(* IEC 61131-3 sources: stc/tests/conveyor, 2 files *)

(* ---- conveyor.st ---- *)
(* Conveyor Belt Control Function Block
   Models a 3-zone conveyor with photoeye sensors, jam detection,
   and state-machine sequencing.

   States:
     0 = IDLE      - Waiting for product
     1 = RUNNING   - Conveyor moving, product in transit
     2 = JAM       - Sensor blocked too long, fault
     3 = STOPPED   - Operator stop requested
*)

FUNCTION_BLOCK ConveyorZone
VAR_INPUT
    Enable      : BOOL;      (* Master enable *)
    SensorEntry : BOOL;      (* Photoeye at zone entry *)
    SensorExit  : BOOL;      (* Photoeye at zone exit *)
    Reset       : BOOL;      (* Reset from jam fault *)
    JamTimeLimit : TIME := T#10s;  (* Max time sensor can be blocked *)
END_VAR

VAR_OUTPUT
    MotorFwd    : BOOL;      (* Drive motor forward *)
    ZoneOccupied : BOOL;     (* Product present in zone *)
    JamFault    : BOOL;      (* Jam detected *)
    State       : INT;       (* Current state *)
    ProductCount : DINT;     (* Products that have exited *)
END_VAR

VAR
    JamTimer    : TON;       (* Jam detection timer *)
    ExitEdge    : R_TRIG;    (* Detects product leaving zone *)
    EntryEdge   : R_TRIG;    (* Detects product entering zone *)
    Counter     : CTU;       (* Product counter *)
END_VAR

    (* Detect product entry and exit edges *)
    EntryEdge(CLK := SensorEntry);
    ExitEdge(CLK := NOT SensorExit);  (* Photoeye: TRUE = blocked *)

    (* State machine *)
    CASE State OF
        0: (* IDLE *)
            MotorFwd := FALSE;
            IF Enable AND SensorEntry THEN
                State := 1;
                ZoneOccupied := TRUE;
            END_IF;

        1: (* RUNNING *)
            MotorFwd := TRUE;
            (* Check for product exit *)
            IF NOT SensorEntry AND NOT SensorExit THEN
                ZoneOccupied := FALSE;
                Counter(CU := TRUE, R := FALSE, PV := 9999);
                State := 0;
            END_IF;
            (* Check for jam *)
            JamTimer(IN := SensorEntry, PT := JamTimeLimit);
            IF JamTimer.Q THEN
                State := 2;
            END_IF;
            IF NOT Enable THEN
                State := 3;
            END_IF;

        2: (* JAM *)
            MotorFwd := FALSE;
            JamFault := TRUE;
            IF Reset THEN
                JamFault := FALSE;
                JamTimer(IN := FALSE, PT := JamTimeLimit);
                State := 0;
            END_IF;

        3: (* STOPPED *)
            MotorFwd := FALSE;
            IF Enable THEN
                State := 1;
            END_IF;
    END_CASE;

    ProductCount := Counter.CV;

    (* Reset counter edge *)
    Counter(CU := FALSE, R := FALSE, PV := 9999);
END_FUNCTION_BLOCK

(* ---- conveyor_test.st ---- *)
(* Conveyor Belt Test Suite
   Tests state machine transitions, jam detection, product counting,
   and enable/disable behavior for a 3-zone conveyor system.
*)

TEST_CASE 'Conveyor starts in IDLE state'
VAR
    State : INT := 0;
    MotorFwd : BOOL := FALSE;
END_VAR
    ASSERT_EQ(State, 0);
    ASSERT_FALSE(MotorFwd);
END_TEST_CASE

TEST_CASE 'Product entry transitions IDLE to RUNNING'
VAR
    State : INT := 0;
    Enable : BOOL := TRUE;
    SensorEntry : BOOL;
    MotorFwd : BOOL;
END_VAR
    (* No product yet *)
    SensorEntry := FALSE;
    CASE State OF
        0:
            MotorFwd := FALSE;
            IF Enable AND SensorEntry THEN
                State := 1;
            END_IF;
    END_CASE;
    ASSERT_EQ(State, 0);
    ASSERT_FALSE(MotorFwd);

    (* Product arrives *)
    SensorEntry := TRUE;
    CASE State OF
        0:
            MotorFwd := FALSE;
            IF Enable AND SensorEntry THEN
                State := 1;
            END_IF;
    END_CASE;
    ASSERT_EQ(State, 1);
END_TEST_CASE

TEST_CASE 'Jam timer triggers fault after timeout'
VAR
    JamTimer : TON;
    SensorEntry : BOOL := TRUE;
    JamFault : BOOL;
END_VAR
    (* Sensor blocked, start timing *)
    JamTimer(IN := SensorEntry, PT := T#10s);
    ASSERT_FALSE(JamTimer.Q);

    (* 8 seconds pass, still no jam *)
    ADVANCE_TIME(T#8s);
    JamTimer(IN := SensorEntry, PT := T#10s);
    ASSERT_FALSE(JamTimer.Q);

    (* 3 more seconds, total 11s > 10s preset *)
    ADVANCE_TIME(T#3s);
    JamTimer(IN := SensorEntry, PT := T#10s);
    ASSERT_TRUE(JamTimer.Q);
    JamFault := JamTimer.Q;
    ASSERT_TRUE(JamFault);
END_TEST_CASE

TEST_CASE 'Jam resets on operator Reset signal'
VAR
    JamTimer : TON;
    JamFault : BOOL := TRUE;
    Reset : BOOL;
    State : INT := 2;
END_VAR
    (* In JAM state, operator presses reset *)
    Reset := TRUE;
    IF Reset THEN
        JamFault := FALSE;
        JamTimer(IN := FALSE, PT := T#10s);
        State := 0;
    END_IF;

    ASSERT_FALSE(JamFault);
    ASSERT_EQ(State, 0);
    ASSERT_FALSE(JamTimer.Q);
END_TEST_CASE

TEST_CASE 'Product counter increments on product exit'
VAR
    Counter : CTU;
END_VAR
    (* Simulate 3 products passing through *)
    Counter(CU := FALSE, R := FALSE, PV := 9999);

    (* Product 1 exits *)
    Counter(CU := TRUE, R := FALSE, PV := 9999);
    ASSERT_EQ(Counter.CV, 1);
    Counter(CU := FALSE, R := FALSE, PV := 9999);

    (* Product 2 exits *)
    Counter(CU := TRUE, R := FALSE, PV := 9999);
    ASSERT_EQ(Counter.CV, 2);
    Counter(CU := FALSE, R := FALSE, PV := 9999);

    (* Product 3 exits *)
    Counter(CU := TRUE, R := FALSE, PV := 9999);
    ASSERT_EQ(Counter.CV, 3);
    ASSERT_FALSE(Counter.Q);  (* PV=9999, far from reached *)
END_TEST_CASE

TEST_CASE 'Disable stops conveyor motor'
VAR
    State : INT := 1;  (* RUNNING *)
    Enable : BOOL;
    MotorFwd : BOOL := TRUE;
END_VAR
    (* Operator disables *)
    Enable := FALSE;

    CASE State OF
        1:
            IF NOT Enable THEN
                State := 3;
                MotorFwd := FALSE;
            END_IF;
    END_CASE;

    ASSERT_EQ(State, 3);
    ASSERT_FALSE(MotorFwd);
END_TEST_CASE

TEST_CASE 'Re-enable resumes from STOPPED to RUNNING'
VAR
    State : INT := 3;  (* STOPPED *)
    Enable : BOOL;
    MotorFwd : BOOL := FALSE;
END_VAR
    Enable := TRUE;
    CASE State OF
        3:
            IF Enable THEN
                State := 1;
            END_IF;
    END_CASE;

    ASSERT_EQ(State, 1);
END_TEST_CASE

TEST_CASE 'Rising edge detects product entry once'
VAR
    EntryEdge : R_TRIG;
    SensorEntry : BOOL;
END_VAR
    (* No product *)
    SensorEntry := FALSE;
    EntryEdge(CLK := SensorEntry);
    ASSERT_FALSE(EntryEdge.Q);

    (* Product arrives: rising edge *)
    SensorEntry := TRUE;
    EntryEdge(CLK := SensorEntry);
    ASSERT_TRUE(EntryEdge.Q);

    (* Product still present: no new edge *)
    EntryEdge(CLK := SensorEntry);
    ASSERT_FALSE(EntryEdge.Q);
END_TEST_CASE
